LIN {X 0,Y 91.941,Z 354.034,A -85,B 0,C 180,E1 -30774.867,E2 -30774.867} C_VEL
LIN {X 0,Y 93.494,Z 341.858,A -85,B 0,C 180,E1 -30775.202,E2 -30775.202} C_VEL
LIN {X 0,Y 92.965,Z 339.573,A -85,B 0,C 180,E1 -30778.376,E2 -30778.376} C_VEL
LIN {X 0,Y 92.686,Z 337.879,A -85,B 0,C 180,E1 -30781.289,E2 -30781.289} C_VEL
LIN {X 0,Y 92.541,Z 337.005,A -85,B 0,C 180,E1 -30784.356,E2 -30784.356} C_VEL
LIN {X 0,Y 92.653,Z 338.294,A -85,B 0,C 180,E1 -30790.547,E2 -30790.547} C_VEL
LIN {X 0,Y 93.374,Z 341.54,A -85,B 0,C 180,E1 -30795.98,E2 -30795.98} C_VEL
LIN {X 0,Y 93.433,Z 341.772,A -85,B 0,C 180,E1 -30796.281,E2 -30796.281} C_VEL
LIN {X 0,Y 91.101,Z 357.793,A -85,B 0,C 180,E1 -30796.848,E2 -30796.848} C_VEL
LIN {X 0,Y 87.965,Z 370.053,A -85,B 0,C 180,E1 -30797.48,E2 -30797.48} C_VEL
LIN {X 0,Y 83.269,Z 382.898,A -85,B 0,C 180,E1 -30798.555,E2 -30798.555} C_VEL
LIN {X 0,Y 77.534,Z 394.713,A -85,B 0,C 180,E1 -30799.92,E2 -30799.92} C_VEL
LIN {X 0,Y 70.865,Z 405.474,A -85,B 0,C 180,E1 -30801.645,E2 -30801.645} C_VEL
LIN {X 0,Y 63.327,Z 415.297,A -85,B 0,C 180,E1 -30803.755,E2 -30803.755} C_VEL
LIN {X 0,Y 55.192,Z 424.195,A -85,B 0,C 180,E1 -30806.997,E2 -30806.997} C_VEL
LIN {X 0,Y 53.369,Z 426.014,A -85,B 0,C 180,E1 -30807.88,E2 -30807.88} C_VEL
LIN {X 0,Y 49.016,Z 429.838,A -85,B 0,C 180,E1 -30809.415,E2 -30809.415} C_VEL
LIN {X 0,Y 37.629,Z 437.715,A -85,B 0,C 180,E1 -30810.635,E2 -30810.635} C_VEL
LIN {X 0,Y 30.907,Z 441.712,A -85,B 0,C 180,E1 -30812.674,E2 -30812.674} C_VEL
LIN {X 0,Y 27.732,Z 443.562,A -85,B 0,C 180,E1 -30815.415,E2 -30815.415} C_VEL
LIN {X 0,Y 18.209,Z 449.039,A -85,B 0,C 180,E1 -30834.68,E2 -30834.68} C_VEL
LIN {X 0,Y 13.118,Z 452.656,A -85,B 0,C 180,E1 -30870.058,E2 -30870.058} C_VEL
LIN {X 0,Y 13.689,Z 454.507,A -85,B 0,C 180,E1 -30900.953,E2 -30900.953} C_VEL
LIN {X 0,Y 22.822,Z 456.912,A -85,B 0,C 180,E1 -30937.567,E2 -30937.567} C_VEL
LIN {X 0,Y 29.16,Z 457.53,A -85,B 0,C 180,E1 -30946.052,E2 -30946.052} C_VEL
LIN {X 0,Y 42.32,Z 457.444,A -85,B 0,C 180,E1 -30955.289,E2 -30955.289} C_VEL
LIN {X 0,Y 55.538,Z 455.876,A -85,B 0,C 180,E1 -30959.999,E2 -30959.999} C_VEL
LIN {X 0,Y 66.838,Z 453.338,A -85,B 0,C 180,E1 -30962.537,E2 -30962.537} C_VEL
LIN {X 0,Y 70.396,Z 452.283,A -85,B 0,C 180,E1 -30963.194,E2 -30963.194} C_VEL
LIN {X 0,Y 70.514,Z 452.314,A -85,B 0,C 180,E1 -30964.608,E2 -30964.608} C_VEL
LIN {X 0,Y 56.686,Z 455.939,A -85,B 0,C 180,E1 -30967.255,E2 -30967.255} C_VEL
LIN {X 0,Y 49.839,Z 457.143,A -85,B 0,C 180,E1 -30969.155,E2 -30969.155} C_VEL
LIN {X 0,Y 36.383,Z 458.329,A -85,B 0,C 180,E1 -30974.963,E2 -30974.963} C_VEL
LIN {X 0,Y 29.89,Z 458.361,A -85,B 0,C 180,E1 -30979.805,E2 -30979.805} C_VEL
LIN {X 0,Y 23.801,Z 458.025,A -85,B 0,C 180,E1 -30987.586,E2 -30987.586} C_VEL
LIN {X 0,Y 14.509,Z 456.115,A -85,B 0,C 180,E1 -31020.971,E2 -31020.971} C_VEL
LIN {X 0,Y 13.201,Z 454.549,A -85,B 0,C 180,E1 -31049.943,E2 -31049.943} C_VEL
LIN {X 0,Y 16.073,Z 451.235,A -85,B 0,C 180,E1 -31090.92,E2 -31090.92} C_VEL
LIN {X 0,Y 23.636,Z 446.806,A -85,B 0,C 180,E1 -31113.046,E2 -31113.046} C_VEL
LIN {X 0,Y 32.965,Z 441.169,A -85,B 0,C 180,E1 -31123.513,E2 -31123.513} C_VEL
LIN {X 0,Y 42.849,Z 434.081,A -85,B 0,C 180,E1 -31129.643,E2 -31129.643} C_VEL
LIN {X 0,Y 53.078,Z 425.225,A -85,B 0,C 180,E1 -31133.083,E2 -31133.083} C_VEL
LIN {X 0,Y 61.679,Z 416.099,A -85,B 0,C 180,E1 -31135.351,E2 -31135.351} C_VEL
LIN {X 0,Y 69.5,Z 406.093,A -85,B 0,C 180,E1 -31136.646,E2 -31136.646} C_VEL
LIN {X 0,Y 76.476,Z 394.946,A -85,B 0,C 180,E1 -31137.596,E2 -31137.596} C_VEL
LIN {X 0,Y 82.593,Z 382.418,A -85,B 0,C 180,E1 -31138.33,E2 -31138.33} C_VEL
LIN {X 0,Y 87.271,Z 369.434,A -85,B 0,C 180,E1 -31138.782,E2 -31138.782} C_VEL
LIN {X 0,Y 90.537,Z 355.743,A -85,B 0,C 180,E1 -31139.212,E2 -31139.212} C_VEL
LIN {X 0,Y 91.905,Z 346.417,A -85,B 0,C 180,E1 -31139.448,E2 -31139.448} C_VEL
LIN {X 0,Y 91.676,Z 344.487,A -85,B 0,C 180,E1 -31143.236,E2 -31143.236} C_VEL
LIN {X 0,Y 91.633,Z 344.144,A -85,B 0,C 180,E1 -31145.252,E2 -31145.252} C_VEL
LIN {X 0,Y 91.721,Z 345.464,A -85,B 0,C 180,E1 -31150.208,E2 -31150.208} C_VEL
LIN {X 0,Y 91.858,Z 346.544,A -85,B 0,C 180,E1 -31152.086,E2 -31152.086} C_VEL
LIN {X 0,Y 89.523,Z 360.208,A -85,B 0,C 180,E1 -31152.481,E2 -31152.481} C_VEL
LIN {X 0,Y 85.807,Z 373.355,A -85,B 0,C 180,E1 -31153.065,E2 -31153.065} C_VEL
LIN {X 0,Y 81.33,Z 384.731,A -85,B 0,C 180,E1 -31153.847,E2 -31153.847} C_VEL
LIN {X 0,Y 75.413,Z 396.213,A -85,B 0,C 180,E1 -31154.847,E2 -31154.847} C_VEL
LIN {X 0,Y 67.709,Z 407.907,A -85,B 0,C 180,E1 -31156.295,E2 -31156.295} C_VEL
LIN {X 0,Y 60.824,Z 416.395,A -85,B 0,C 180,E1 -31157.647,E2 -31157.647} C_VEL
LIN {X 0,Y 52.359,Z 425.167,A -85,B 0,C 180,E1 -31160.075,E2 -31160.075} C_VEL
LIN {X 0,Y 43.984,Z 432.411,A -85,B 0,C 180,E1 -31163.31,E2 -31163.31} C_VEL
LIN {X 0,Y 34.184,Z 439.536,A -85,B 0,C 180,E1 -31169.155,E2 -31169.155} C_VEL
LIN {X 0,Y 27.732,Z 443.562,A -85,B 0,C 180,E1 -31175.415,E2 -31175.415} C_VEL
LIN {X 0,Y 22.919,Z 446.17,A -85,B 0,C 180,E1 -31180.509,E2 -31180.509} C_VEL
LIN {X 0,Y 14.236,Z 449.887,A -85,B 0,C 180,E1 -31190.223,E2 -31190.223} C_VEL
LIN {X 0,Y 7.774,Z 452.385,A -85,B 0,C 180,E1 -31212.424,E2 -31212.424} C_VEL
LIN {X 0,Y 6.166,Z 453.999,A -85,B 0,C 180,E1 -31259.447,E2 -31259.447} C_VEL
LIN {X 0,Y 6.944,Z 454.445,A -85,B 0,C 180,E1 -31274.938,E2 -31274.938} C_VEL
LIN {X 0,Y 14.382,Z 456.359,A -85,B 0,C 180,E1 -31308.006,E2 -31308.006} C_VEL
LIN {X 0,Y 27.155,Z 457.834,A -85,B 0,C 180,E1 -31319.999,E2 -31319.999} C_VEL
LIN {X 0,Y 35.208,Z 458.006,A -85,B 0,C 180,E1 -31323.307,E2 -31323.307} C_VEL
LIN {X 0,Y 35.223,Z 458.016,A -85,B 0,C 180,E1 -31323.69,E2 -31323.69} C_VEL
LIN {X 0,Y 28.282,Z 458.017,A -85,B 0,C 180,E1 -31326.092,E2 -31326.092} C_VEL
LIN {X 0,Y 21.451,Z 457.632,A -85,B 0,C 180,E1 -31330.451,E2 -31330.451} C_VEL
LIN {X 0,Y 8.981,Z 455.649,A -85,B 0,C 180,E1 -31358.374,E2 -31358.374} C_VEL
LIN {X 0,Y 6.112,Z 454.053,A -85,B 0,C 180,E1 -31409.876,E2 -31409.876} C_VEL
LIN {X 0,Y 11.66,Z 450.669,A -85,B 0,C 180,E1 -31474.544,E2 -31474.544} C_VEL
LIN {X 0,Y 21.368,Z 446.167,A -85,B 0,C 180,E1 -31490.4,E2 -31490.4} C_VEL
LIN {X 0,Y 31.685,Z 440.451,A -85,B 0,C 180,E1 -31496.043,E2 -31496.043} C_VEL
LIN {X 0,Y 42.153,Z 433.225,A -85,B 0,C 180,E1 -31499.342,E2 -31499.342} C_VEL
LIN {X 0,Y 52.697,Z 424.271,A -85,B 0,C 180,E1 -31500.826,E2 -31500.826} C_VEL
LIN {X 0,Y 61.515,Z 415.012,A -85,B 0,C 180,E1 -31502.056,E2 -31502.056} C_VEL
LIN {X 0,Y 69.448,Z 404.797,A -85,B 0,C 180,E1 -31502.502,E2 -31502.502} C_VEL
LIN {X 0,Y 75.627,Z 395.001,A -85,B 0,C 180,E1 -31502.894,E2 -31502.894} C_VEL
LIN {X 0,Y 81.81,Z 382.568,A -85,B 0,C 180,E1 -31503.241,E2 -31503.241} C_VEL
LIN {X 0,Y 86.327,Z 370.478,A -85,B 0,C 180,E1 -31503.436,E2 -31503.436} C_VEL
LIN {X 0,Y 89.683,Z 357.295,A -85,B 0,C 180,E1 -31503.687,E2 -31503.687} C_VEL
LIN {X 0,Y 90.702,Z 351.44,A -85,B 0,C 180,E1 -31503.889,E2 -31503.889} C_VEL
LIN {X 0,Y 90.652,Z 351.439,A -85,B 0,C 180,E1 -31506.121,E2 -31506.121} C_VEL
LIN {X 0,Y 90.641,Z 351.795,A -85,B 0,C 180,E1 -31507.684,E2 -31507.684} C_VEL
LIN {X 0,Y 88.054,Z 364.3,A -85,B 0,C 180,E1 -31508.03,E2 -31508.03} C_VEL
LIN {X 0,Y 84.138,Z 376.59,A -85,B 0,C 180,E1 -31508.464,E2 -31508.464} C_VEL
LIN {X 0,Y 79.118,Z 388.185,A -85,B 0,C 180,E1 -31509.041,E2 -31509.041} C_VEL
LIN {X 0,Y 73.044,Z 399.094,A -85,B 0,C 180,E1 -31509.618,E2 -31509.618} C_VEL
LIN {X 0,Y 66.071,Z 409.166,A -85,B 0,C 180,E1 -31510.381,E2 -31510.381} C_VEL
LIN {X 0,Y 59.066,Z 417.493,A -85,B 0,C 180,E1 -31511.097,E2 -31511.097} C_VEL
LIN {X 0,Y 50.371,Z 426.134,A -85,B 0,C 180,E1 -31512.493,E2 -31512.493} C_VEL
LIN {X 0,Y 39.96,Z 434.523,A -85,B 0,C 180,E1 -31514.787,E2 -31514.787} C_VEL
LIN {X 0,Y 29.635,Z 441.276,A -85,B 0,C 180,E1 -31518.544,E2 -31518.544} C_VEL
LIN {X 0,Y 19.481,Z 446.681,A -85,B 0,C 180,E1 -31525.693,E2 -31525.693} C_VEL
LIN {X 0,Y 10.042,Z 450.92,A -85,B 0,C 180,E1 -31545.694,E2 -31545.694} C_VEL
LIN {X 0,Y 5.902,Z 453.199,A -85,B 0,C 180,E1 -31590.128,E2 -31590.128} C_VEL
LIN {X 0,Y 6.944,Z 454.445,A -85,B 0,C 180,E1 -31634.938,E2 -31634.938} C_VEL
LIN {X 0,Y 7.883,Z 456.385,A -85,B 0,C 180,E1 -31644.162,E2 -31644.162} C_VEL
LIN {X 0,Y 7.883,Z 600,A -85,B 0,C 180,E1 -31644.162,E2 -31644.162} C_VEL
LIN {X 0,Y 7.883,Z 600,A -85,B 0,C 180,E1 -31644.162,E2 -31644.162}

QRS_NEXT_CUT()

QRS_NEXT()
QRS_HOME()

END
